TYPE MIS_PC :
STRUCT
	Step_PC       : ARRAY[0..MAX_STEP_MISS] OF Step_PC;	// Array step programma  (0..500)
	Tot_step_PC	  : UINT;						// Numero di steps della missione
	Pstart_PC     : UINT;						// Nodo iniziale missione (=Nodo attuale ASRV)
	Pend_PC       : UINT;						// Nodo fine missione (eventuale di carico/scarico)
	Typ_car_PC    : UINT;						// Tipo di stabilità carico (0 massima, 9 minima)
	MisFree1      : UINT;
	MisFree2      : UINT;
	MisFree3      : UINT;
END_STRUCT
END_TYPE

(* stored: Version 1.1.0.1, ProductVersion 3.1.4024.11
   DUT MIS_PC: Id {41e9883d-5ed0-4350-94a0-cac9995f1bc3} *)
